// TIA Portal V19 export
TYPE "Positioning_DOL_Machine_Alr"
// stored: Access Published
   STRUCT
      Ax : "OOAx_Alr";   // ON-OFF AXIS
      Ax_NotHomed : Bool;   // Axis not homed / referenced
      S120 : Struct   // SINAMICS S120
         Drive { ExternalAccessible := 'False'; ExternalVisible := 'False'; ExternalWritable := 'False'} : Bool;   // warning presence
      END_STRUCT;
      S120_ComErr : Bool;   // Interruption of communication to the SINAMICS drive
      BrakeTimeOut : Bool;   // Brake feedback timeout
      Fan_M : "MotorAlr";   // MOTOR FAN
   END_STRUCT;
END_TYPE
